{attribute addProperty BoxType "EL3061-0000-0017"}
{attribute addProperty Id "AI_StandardAT %I*AI_Standard_B51B79FC8110.1250WcStateAT %I*WcState_98A4DF7520.250InfoDataAT %I*InfoData_BC63D37F80100"}
{attribute addProperty CRC "1285133446"}
{attribute addProperty SizeInBites "163"}
{attribute addProperty SizeInBytes "20.375"}
TYPE EL3061_639E8231 :
STRUCT
	{attribute addProperty Name "AI_Standard"}
	AI_Standard : AI_Standard_B51B79FC;
	{attribute addProperty Name "WcState"}
	WcState : WcState_98A4DF75;
	{attribute addProperty Name "InfoData"}
	InfoData : InfoData_BC63D37F;
END_STRUCT
END_TYPE

(* stored: Version 1.2.0.0, ProductVersion 3.1.4024.9
   DUT EL3061_639E8231: Id {0ff4c9d7-3b72-43ef-88ff-73e56ef5c363} *)
